Universal Robots PolyScope program: orange_Bridge_triangle_roof.urp

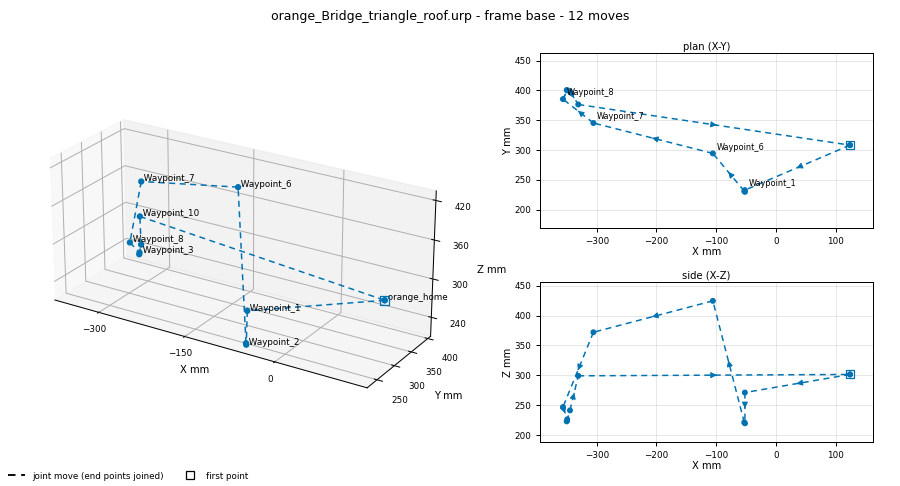
[picture p0: tool path of orange_Bridge_triangle_roof.urp in frame base, 12 of 12 moves have a stored position in this frame; points joined in program order, loops and branches not executed]
Program orange_Bridge_triangle_roof (installation=default directory=/programs/usbdisk/Zahra1/orangi createdIn=5.11.11.1010533 lastSavedIn=5.11.11.1010533 robotSerialNumber=20205300864)
Calibrated DH parameters: a=[-0.000166, -0.243494, -0.153108, 0.000057, -0.000123, 0]; d=[0.151897, -1.34267, 53.988124, -52.514559, 0.085283, 0.092193]; alpha=[1.572472, -0.003756, 0.002824, 1.570807, -1.572621, 0]; deltaTheta=[0, 0.020704, 7.033215, -0.770746, 0.000004, 0]
Robot Program (runOnlyOnce=true)
  MoveJ speed 60 deg/s, acceleration 80 deg/s^2 (useActiveTCP=true) feature=Base
    Waypoint orange_home: TCP in base x=124.286 y=308.277 z=301.462 mm, rx=2.2499 ry=-2.1846 rz=-0.0963 rad; joints [-269.66, -91.226, -90.279, -86.086, 92.69, 808.818] deg
    Waypoint Waypoint_1: TCP in base x=-51.906 y=232.915 z=271.119 mm, rx=2.3171 ry=-2.0857 rz=0.0246 rad; joints [-224.897, -66.866, -116.254, -87.746, 91.44, 849.163] deg
    URCap Gripper (Robotiq_Grippers, Robotiq Inc.) dataModel(position=27.058823529411764, force=94.0, speed=28.0, positionInDouble=27.058823529411764, forceInDouble=94.0, speedInDouble=28.0, slaveIds=[9], blocking=true, robotCompliant=false)
    Waypoint Waypoint_2: TCP in base x=-51.748 y=230.03 z=219.621 mm, rx=2.2148 ry=-2.178 rz=-0.036 rad; joints [-224.672, -68.031, -130.698, -69.837, 92.145, 854.526] deg
    URCap Gripper (Robotiq_Grippers, Robotiq Inc.) dataModel(position=59.2156862745098, force=94.0, speed=40.0, positionInDouble=59.2156862745098, forceInDouble=94.0, speedInDouble=40.0, slaveIds=[9], blocking=true, robotCompliant=false)
    Waypoint Waypoint_5: TCP in base x=-52.922 y=231.258 z=221.198 mm, rx=2.2045 ry=-2.1894 rz=-0.0274 rad; joints [-224.668, -68.466, -129.875, -70.533, 92.104, 855.091] deg
    Waypoint Waypoint_6: TCP in base x=-105.539 y=294.437 z=424.762 mm, rx=-2.1548 ry=2.2231 rz=0.0863 rad; joints [-224.704, -93.161, -53.618, -119.976, 87.323, 857.061] deg
    Waypoint Waypoint_7: TCP in base x=-305.688 y=345.334 z=372.113 mm, rx=2.1904 ry=-2.2331 rz=-0.2722 rad; joints [-211.464, -131.613, -15.831, -112.773, 87.488, 869.415] deg
    Waypoint Waypoint_8: TCP in base x=-356.663 y=385.366 z=246.849 mm, rx=-2.1692 ry=2.2184 rz=0.1335 rad; joints [-212.184, -149.383, -15.257, -100.937, 86.654, 868.937] deg
    Waypoint Waypoint_3: TCP in base x=-349.474 y=400.091 z=226.171 mm, rx=2.1786 ry=-2.2137 rz=-0.0951 rad; joints [-214.803, -152.931, -13.523, -99.631, 91.08, 866.11] deg
    Waypoint Waypoint_9: TCP in base x=-350.337 y=400.572 z=222.853 mm, rx=2.1785 ry=-2.2134 rz=-0.0919 rad; joints [-214.8, -153.328, -13.576, -99.295, 91.121, 866.107] deg
    URCap Gripper (Robotiq_Grippers, Robotiq Inc.) dataModel(position=33.72549019607843, force=94.0, speed=40.0, positionInDouble=33.72549019607843, forceInDouble=94.0, speedInDouble=40.0, slaveIds=[9], blocking=true, robotCompliant=false)
    Waypoint Waypoint_4: TCP in base x=-344.906 y=398.157 z=241.241 mm, rx=2.1992 ry=-2.2033 rz=-0.125 rad; joints [-214.805, -150.218, -15.305, -99.582, 90.455, 865.288] deg
    Waypoint Waypoint_10: TCP in base x=-331.017 y=376.377 z=299.134 mm, rx=-2.2399 ry=2.1889 rz=0.1197 rad; joints [-213.243, -145.317, -8.373, -111.99, 88.522, 865.347] deg
    Waypoint orange_home: TCP in base x=124.286 y=308.277 z=301.462 mm, rx=2.2499 ry=-2.1846 rz=-0.0963 rad; joints [-269.66, -91.226, -90.279, -86.086, 92.69, 808.818] deg
